FUNCTION_BLOCK FB_RecipeBase EXTENDS FB_PackML_BaseModule IMPLEMENTS I_RecipeBuilder

VAR
    RecipeBuilder_HMI		: ST_RecipeBuilder_HMI;
    _Config                 : ST_RecipeBuilder_Config;
    _PanelFrontLength       : REAL;  
    _PanelFrontWidth        : REAL;      
    _PanelHeight            : REAL;    
    _RailHeightCorrection   : REAL;

    // --- NOWE ZMIENNE DO PRZECHOWYWANIA SEGMENTÓW ---
    _SegmentsCutX           : ARRAY [1..32] OF ST_CutSegment;
    _SegmentsCutY           : ARRAY [1..32] OF ST_CutSegment;
    _SegmentsGroove         : ARRAY [1..32] OF ST_CutSegment;
    _SegmentsToCutX         : INT;
    _SegmentsToCutY         : INT;
    _SegmentsToGroove       : INT;
END_VAR

METHOD Build : BOOL
Build := FALSE;
END_METHOD

PROPERTY Config : ST_RecipeBuilder_Config
GET
Config := _Config;
END_GET
SET
_Config := Config;
RecipeBuilder_HMI.Config := Config;
END_SET
END_PROPERTY

// Provides interlocks for HMI control and updates HMI status information for this module
METHOD PROTECTED HMICommunication

// This method is called cyclically by CyclicLogic()
// Zamiast przepisywać do rozbitych zmiennych (_PanelFrontWidth itp.),
// zaktualizuj całą strukturę wewnętrzną:
_Config := RecipeBuilder_HMI.Config;

// Przypisania do rozbitych zmiennych możesz zachować, jeśli używasz ich gdzieś indziej,
// ale _Config jest kluczowy dla metody Build().
_PanelFrontWidth      := RecipeBuilder_HMI.Config.PanelFrontWidht;
_PanelFrontLength     := RecipeBuilder_HMI.Config.PanelFrontLength;
_PanelHeight          := RecipeBuilder_HMI.Config.PanelHeight;
_RailHeightCorrection := RecipeBuilder_HMI.Config.RailHeightCorrection;
END_METHOD

PROPERTY SegmentsCutX : REFERENCE TO ARRAY [1..32] OF ST_CutSegment
GET
SegmentsCutX REF= _SegmentsCutX;
END_GET
END_PROPERTY

PROPERTY SegmentsCutY : REFERENCE TO ARRAY [1..32] OF ST_CutSegment
GET
SegmentsCutY REF= _SegmentsCutY;
END_GET
END_PROPERTY

PROPERTY SegmentsGroove : REFERENCE TO ARRAY [1..32] OF ST_CutSegment
GET
SegmentsGroove REF= _SegmentsGroove;
END_GET
END_PROPERTY


PROPERTY SegmentsToCutX : INT
GET
SegmentsToCutX := _SegmentsToCutX;
END_GET
END_PROPERTY


PROPERTY SegmentsToCutY : INT
GET
SegmentsToCutY := _SegmentsToCutY;
END_GET
END_PROPERTY


PROPERTY SegmentsToGroove : INT
GET
SegmentsToGroove := _SegmentsToGroove;
END_GET
END_PROPERTY

END_FUNCTION_BLOCK

(* stored: Version 1.1.0.1, ProductVersion 3.1.4024.15
   POU FB_RecipeBase: Id {da96ec31-8163-452f-a094-4558fa21ef5c}, SpecialFunc None
   Method Build: Id {47409b61-265d-42e6-ab22-9bedebae5b88}
   Property Config: Id {cc8b22ea-aed1-438f-8cdd-5e3e5f7b2e90}
   Get Get: Id {51a4be92-27e0-4d30-897e-f466d704a9e2}
   Set Set: Id {ea17f2c2-4fb3-4cd4-85eb-6bcadc1e2873}
   Method HMICommunication: Id {9b128247-8dae-407e-a375-ac93c0194d56}
   Property SegmentsCutX: Id {3184be54-f03a-4975-8cf1-db07c128d253}
   Get Get: Id {0f425160-36a8-4f28-99b9-e92bc5ef61d9}
   Property SegmentsCutY: Id {7e96d748-34eb-4d02-bea9-39c6162fca26}
   Get Get: Id {18ebbd77-7872-47d5-b7ea-e1c19856104e}
   Property SegmentsGroove: Id {ef32f872-b41e-411a-89df-3b90001a16fb}
   Get Get: Id {9f573555-28d1-42d5-8de5-c6e1c98b00d0}
   Property SegmentsToCutX: Id {7c141887-7a79-44a8-a421-fb9ee098c25b}
   Get Get: Id {549e99d8-5984-4542-b902-6ce577ebde0d}
   Property SegmentsToCutY: Id {2a1a5acb-e3ff-4cf0-ad15-d0b6b45a1d0e}
   Get Get: Id {4f78cbac-d000-4132-997b-ee432b29e987}
   Property SegmentsToGroove: Id {c7b518f5-2d21-49fc-94c1-1f117859a4b1}
   Get Get: Id {8e366a6f-311d-4e3a-904c-a58ce6da4751} *)
